        // History ring buffer update
        "DB_Production".Hist_Index := "DB_Production".Hist_Index + 1;
        IF "DB_Production".Hist_Index > 100 THEN
            "DB_Production".Hist_Index := 1;
        END_IF;
        IF "DB_Production".Hist_Count < 100 THEN
            "DB_Production".Hist_Count := "DB_Production".Hist_Count + 1;
        END_IF;
        "DB_Production".Hist_Result["DB_Production".Hist_Index] := "DB_Production".LastResult;
        "DB_Production".Hist_Program["DB_Production".Hist_Index] := "DB_Production".LastProgram;
        "DB_Production".Hist_Duration_s["DB_Production".Hist_Index] := "DB_Production".LastDuration_s;
        "DB_Production".Hist_ErrorCode["DB_Production".Hist_Index] := "DB_Production".LastErrorCode;
        "DB_Production".Hist_ErrorLine["DB_Production".Hist_Index] := "DB_Production".LastErrorLine;
        "DB_Production".Hist_Time["DB_Production".Hist_Index] := #prodTimeNow;
    END_IF;

    // Edge: NOK (enter STATE_ERROR with active cycle)
    IF (#State = STATE_ERROR) AND (#prevState <> STATE_ERROR) AND "DB_Production".CurrentActive THEN
        "DB_Production".LastResult := 2;  // NOK
        "DB_Production".LastProgram := #activeProgram;
        "DB_Production".LastDuration_s := "DB_HMI".ElapsedSeconds;
        "DB_Production".LastErrorCode := #fbAlarmManager.ActiveErrorCode;
        "DB_Production".LastErrorLine := "DB_Diagnostic".Error_Line;
        "DB_Production".TotalNOK := "DB_Production".TotalNOK + 1;
        #prodTimeStatus := RD_SYS_T(OUT => #prodTimeNow);
        "DB_Production".LastEndTime := #prodTimeNow;
        "DB_Production".CurrentActive := FALSE;

        // History ring buffer update
        "DB_Production".Hist_Index := "DB_Production".Hist_Index + 1;
        IF "DB_Production".Hist_Index > 100 THEN
            "DB_Production".Hist_Index := 1;
        END_IF;
        IF "DB_Production".Hist_Count < 100 THEN
            "DB_Production".Hist_Count := "DB_Production".Hist_Count + 1;
        END_IF;
        "DB_Production".Hist_Result["DB_Production".Hist_Index] := "DB_Production".LastResult;
        "DB_Production".Hist_Program["DB_Production".Hist_Index] := "DB_Production".LastProgram;
        "DB_Production".Hist_Duration_s["DB_Production".Hist_Index] := "DB_Production".LastDuration_s;
        "DB_Production".Hist_ErrorCode["DB_Production".Hist_Index] := "DB_Production".LastErrorCode;
        "DB_Production".Hist_ErrorLine["DB_Production".Hist_Index] := "DB_Production".LastErrorLine;
        "DB_Production".Hist_Time["DB_Production".Hist_Index] := #prodTimeNow;
    END_IF;

    // Edge: STOPPED via STOP sequence (STOPPING / STOP_GOHOME / STOP_GOTOZERO → STOPPED)
    IF (#State = STATE_STOPPED) AND
       ((#prevState = STATE_STOPPING) OR (#prevState = STATE_STOP_GOHOME) OR (#prevState = STATE_STOP_GOTOZERO)) AND
       "DB_Production".CurrentActive THEN
        "DB_Production".LastResult := 3;  // STOP
        "DB_Production".LastProgram := #activeProgram;
        "DB_Production".LastDuration_s := "DB_HMI".ElapsedSeconds;
        "DB_Production".LastErrorCode := 0;
        "DB_Production".LastErrorLine := -1;
        "DB_Production".TotalStopped := "DB_Production".TotalStopped + 1;
        #prodTimeStatus := RD_SYS_T(OUT => #prodTimeNow);
        "DB_Production".LastEndTime := #prodTimeNow;
        "DB_Production".CurrentActive := FALSE;

        // History ring buffer update
        "DB_Production".Hist_Index := "DB_Production".Hist_Index + 1;
        IF "DB_Production".Hist_Index > 100 THEN
            "DB_Production".Hist_Index := 1;
        END_IF;
        IF "DB_Production".Hist_Count < 100 THEN
            "DB_Production".Hist_Count := "DB_Production".Hist_Count + 1;
        END_IF;
        "DB_Production".Hist_Result["DB_Production".Hist_Index] := "DB_Production".LastResult;
        "DB_Production".Hist_Program["DB_Production".Hist_Index] := "DB_Production".LastProgram;
        "DB_Production".Hist_Duration_s["DB_Production".Hist_Index] := "DB_Production".LastDuration_s;
        "DB_Production".Hist_ErrorCode["DB_Production".Hist_Index] := "DB_Production".LastErrorCode;
        "DB_Production".Hist_ErrorLine["DB_Production".Hist_Index] := "DB_Production".LastErrorLine;
        "DB_Production".Hist_Time["DB_Production".Hist_Index] := #prodTimeNow;
    END_IF;

    // Production RESET: clear counters + history
    IF #prodResetEdge THEN
        "DB_Production".TotalStarted := 0;
        "DB_Production".TotalOK := 0;
        "DB_Production".TotalNOK := 0;
        "DB_Production".TotalStopped := 0;
        "DB_Production".Hist_Index := 0;
        "DB_Production".Hist_Count := 0;
        // Optionally also clear last cycle summary
        "DB_Production".LastResult := 0;
        "DB_Production".LastProgram := 0;
        "DB_Production".LastDuration_s := 0;
        "DB_Production".LastErrorCode := 0;
        "DB_Production".LastErrorLine := -1;
        "DB_Production".CurrentActive := FALSE;
    END_IF;

    // Last-cycle RESET: only clear last cycle summary (counters and history are preserved)
    IF #lastCycleResetEdge THEN
        "DB_Production".LastResult := 0;
        "DB_Production".LastProgram := 0;
        "DB_Production".LastDuration_s := 0;
        "DB_Production".LastErrorCode := 0;
        "DB_Production".LastErrorLine := -1;
    END_IF;

    // Update prevState for next cycle
    #prevState := #State;

    // =========================================================================
    // RECIPE HANDLER - Execute based on active program
    // =========================================================================
    CASE #activeProgram OF
        1: #fbRecipeHandler(Start := #bStartSeq, Stop := #fbInputs.Cmd_Stop,
                            Pause := #bPauseActive, Reset := #fbInputs.Cmd_Reset OR #bResetRecipe,
                            StartLine := MAX(IN1:= INT#0, IN2:= #savedLineIndex),
                            LineCount := #activeLineCount,
                            Lines := "DB_RecipeProgram1".Lines,
                            Axis_X := #Axis_X, Axis_Z := #Axis_Z);
        2: #fbRecipeHandler(Start := #bStartSeq, Stop := #fbInputs.Cmd_Stop,
                            Pause := #bPauseActive, Reset := #fbInputs.Cmd_Reset OR #bResetRecipe,
                            StartLine := MAX(IN1:= INT#0,IN2:= #savedLineIndex),
                            LineCount := #activeLineCount,
                            Lines := "DB_RecipeProgram2".Lines,
                            Axis_X := #Axis_X, Axis_Z := #Axis_Z);
        3: #fbRecipeHandler(Start := #bStartSeq, Stop := #fbInputs.Cmd_Stop,
                            Pause := #bPauseActive, Reset := #fbInputs.Cmd_Reset OR #bResetRecipe,
                            StartLine := MAX(IN1:= INT#0,IN2:= #savedLineIndex),
                            LineCount := #activeLineCount,
                            Lines := "DB_RecipeProgram3".Lines,
                            Axis_X := #Axis_X, Axis_Z := #Axis_Z);
        4: #fbRecipeHandler(Start := #bStartSeq, Stop := #fbInputs.Cmd_Stop,
                            Pause := #bPauseActive, Reset := #fbInputs.Cmd_Reset OR #bResetRecipe,
                            StartLine := MAX(IN1:= INT#0,IN2:= #savedLineIndex),
                            LineCount := #activeLineCount,
                            Lines := "DB_RecipeProgram4".Lines,
                            Axis_X := #Axis_X, Axis_Z := #Axis_Z);
        5: #fbRecipeHandler(Start := #bStartSeq, Stop := #fbInputs.Cmd_Stop,
                            Pause := #bPauseActive, Reset := #fbInputs.Cmd_Reset OR #bResetRecipe,
                            StartLine := MAX(IN1:= INT#0,IN2:= #savedLineIndex),
                            LineCount := #activeLineCount,
                            Lines := "DB_RecipeProgram5".Lines,
                            Axis_X := #Axis_X, Axis_Z := #Axis_Z);
    END_CASE;

    // Homing -- sequential pattern: STATE_HOMING (startup) and STATE_STOP_GOHOME (post-stop)
    // both use homeSeqState + bHomeXExec/bHomeZExec.
    // Mode SEL: mode 3 (active+zero) is forced in STATE_HOMING; other states use DB_Manual.HomingMode.
    #fbHomeX(
        Execute := #bHomeXExec,
        Mode := SEL(G := (#State = STATE_HOMING AND #bHomeXExec), IN0 := 3, IN1 := "DB_Manual".HomingMode),
        Position := "DB_MachineConfig".HomeOffset_X,
        Axis := #Axis_X
    );
    #fbHomeZ(
        Execute := #bHomeZExec,
        Mode := SEL(G := (#State = STATE_HOMING AND #bHomeZExec), IN0 := 3, IN1 := "DB_Manual".HomingMode),
        Position := "DB_MachineConfig".HomeOffset_Z,
        Axis := #Axis_Z
    );
    #fbHomeTool(
        Execute  := #bHomeToolExec,
        Mode     := SEL(G := (#State = STATE_HOMING AND #bHomeToolExec), IN0 := 3, IN1 := "DB_Manual".HomingMode),
        Position := 0.0,
        Axis     := #Axis_Tool
    );
    // PNP halt FBs: Execute stays TRUE until bHaltX/Z_PNP is cleared (on return to STATE_STOPPED)
    #fbHaltX_PNP(Execute := #bHaltX_PNP, Axis := #Axis_X);
    #fbHaltZ_PNP(Execute := #bHaltZ_PNP, Axis := #Axis_Z);

    // Tool changer -- only rotates the turret; axis positioning done by G-code
    #fbToolChanger(Execute := #bToolExecute, ToolNumber := #activeToolReq,
                   Axis_Tool := #Axis_Tool);

    // Motion FBs for moving to position 0 after stop
    #fbMoveX_Stop(Execute := #bStopMoveX, Position := 0.0, Velocity := "DB_MachineConfig".RapidVelocity, Axis := #Axis_X);
    #fbMoveZ_Stop(Execute := #bStopMoveZ, Position := 0.0, Velocity := "DB_MachineConfig".RapidVelocity, Axis := #Axis_Z);
    // Homing clearance moves -- pre (clear PNP zone) and post (move away after homing)
    // Target: HomeOffset + PostHome_Clearance (outside PNP sensor range)
    #fbMoveX_HomeClr(Execute  := #bHomeClrX,
                     Position := "DB_MachineConfig".HomeOffset_X + "DB_MachineConfig".PostHome_Clearance,
                     Velocity := "DB_MachineConfig".HomeVelocity,
                     Axis     := #Axis_X);
    #fbMoveZ_HomeClr(Execute  := #bHomeClrZ,
                     Position := "DB_MachineConfig".HomeOffset_Z + "DB_MachineConfig".PostHome_Clearance,
                     Velocity := "DB_MachineConfig".HomeVelocity,
                     Axis     := #Axis_Z);

    // Manual mode - sync aliases first
    // In STATE_PNP_HALT: block jog direction that would drive the axis deeper into the PNP zone.
    // Jog toward the active PNP zone is blocked; jog away (escape direction) is passed through.
    IF #State = STATE_PNP_HALT THEN
        "DB_Manual".Jog_Plus  := "DB_Manual".Btn_JogPlus AND NOT (
            ("DB_Manual".SelectedAxis = 0 AND #HW_PNP_X_Max) OR
            ("DB_Manual".SelectedAxis = 1 AND #HW_PNP_Z_Max));
        "DB_Manual".Jog_Minus := "DB_Manual".Btn_JogMinus AND NOT (
            ("DB_Manual".SelectedAxis = 0 AND #HW_PNP_X_Min) OR
            ("DB_Manual".SelectedAxis = 1 AND #HW_PNP_Z_Min));
    ELSE
        "DB_Manual".Jog_Plus  := "DB_Manual".Btn_JogPlus;
        "DB_Manual".Jog_Minus := "DB_Manual".Btn_JogMinus;
    END_IF;
    "DB_Manual".Btn_HomeAxis := "DB_Manual".Btn_Home;

    #fbManualMode(Enable := (#State = STATE_MANUAL OR #State = STATE_PNP_HALT),
                  SelectedAxis := "DB_Manual".SelectedAxis,
                  Jog_Plus := "DB_Manual".Jog_Plus, Jog_Minus := "DB_Manual".Jog_Minus,
                  JogSpeed := "DB_Manual".JogSpeed,
                  MoveAbsolute := "DB_Manual".Btn_MoveAbsolute, TargetPosition := "DB_Manual".MoveToPosition,
                  HomeAxis := "DB_Manual".Btn_HomeAxis, HomeAll := "DB_Manual".Btn_HomeAll,
                  HomingMode := "DB_Manual".HomingMode, HomePosition := 0.0,
                  GoSafe := "DB_Manual".Btn_GoSafe, GoZero := "DB_Manual".Btn_GoZero,
                  SafeToJog := #fbSafetyMonitor.SafeToJog, Reset := #fbInputs.Cmd_Reset,
                  PNP_X_Min := #HW_PNP_X_Min, PNP_Z_Min := #HW_PNP_Z_Min,
                  ToolStepCW := "DB_Manual".Btn_ToolStepCW, ToolStepCCW := "DB_Manual".Btn_ToolStepCCW,
                  ToolStepAngle := "DB_Manual".ToolStepAngle, ToolStepSpeed := "DB_Manual".ToolStepSpeed,
                  Axis_X := #Axis_X, Axis_Z := #Axis_Z, Axis_Tool := #Axis_Tool, Axis_Spindle := #Axis_Spindle);

    // Update manual mode status
    "DB_Manual".JogBusy := #fbManualMode.Busy;
    "DB_Manual".ManualBusy := #fbManualMode.Busy;       // Alias
    "DB_Manual".JogError := #fbManualMode.Error;
    "DB_Manual".ManualError := #fbManualMode.Error;     // Alias
    "DB_Manual".JogErrorID := #fbManualMode.ErrorID;
    "DB_Manual".ManualErrorID := #fbManualMode.ErrorID; // Alias
    "DB_Manual".SelectedAxisPos := SEL(G := "DB_Manual".SelectedAxis = 0,
                                        IN0 := #Axis_Z.ActualPosition, IN1 := #Axis_X.ActualPosition);
    "DB_Manual".SelectedAxisName := SEL(G := "DB_Manual".SelectedAxis = 0, IN0 := 'Z', IN1 := 'X');
    "DB_Manual".ToolPosition := #Axis_Tool.ActualPosition;
    "DB_Manual".ActiveAxis := #fbManualMode.ActiveAxis;

    // Forward manual mode errors to alarm manager (once, on rising edge)
    IF #fbManualMode.Error AND NOT #prevManualError THEN
        #newErrorFlag := TRUE;
        #newErrorCode := #fbManualMode.ErrorID;
        // DB_HMI.ErrorDetail is written directly inside FB_ManualMode at each error point.
        // Write ErrorText here as a fallback for any code not yet handled with direct detail.
        "DB_HMI".ErrorText := 'Manual mode error - check ErrorDetail and ErrorID';
    END_IF;
    #prevManualError := #fbManualMode.Error;

    // =========================================================================
    // SPINDLE CONTROL
    // Manual mode spindle control via DB_Manual buttons
    // Recipe handler spindle control via bSpindleStart/bSpindleStop flags
    // =========================================================================
    #fbSpindleControl(
        Enable := #bDrivesEnable,  // Drive stays powered during normal operation; cut on E-Stop or STATE_ERROR
        Start := "DB_Manual".Btn_SpindleStart OR #bSpindleStart,
        Stop := "DB_Manual".Btn_SpindleStop OR #bSpindleStop OR #fbInputs.Cmd_Stop,
        SetSpeed := SEL(G := (#State = STATE_MANUAL),
                        IN0 := "DB_Spindle".Cmd_SetSpeed,
                        IN1 := "DB_Manual".Manual_SpindleSpeed),
        Direction := SEL(G := (#State = STATE_MANUAL),
                         IN0 := "DB_Spindle".Cmd_Direction,
                         IN1 := "DB_Manual".Manual_SpindleDir),
        SpeedOverride := "DB_Spindle".SpeedOverride,
        Reset := #fbInputs.Cmd_Reset OR #bResetRecipe,  // Also reset on recipe restart (clears state 999 error)
        AckError := #ackEdge OR "DB_Manual".Btn_SpindleAckError,  // Main Ack or spindle-specific Ack (no full Reset needed)
        Axis_Spindle := #Axis_Spindle
    );

    // Diagnostic output
    "DB_Diagnostic".Process_State        := #State;
    "DB_Diagnostic".Process_SafeToRun    := #SafeToRun;
    "DB_Diagnostic".Process_DrivesEnable := #bDrivesEnable;
    "DB_Diagnostic".Recipe_CurrentProgram := #activeProgram;
    "DB_Diagnostic".Recipe_TotalLines    := #activeLineCount;
    "DB_Diagnostic".Axis_X_Pos           := #Axis_X.ActualPosition;
    "DB_Diagnostic".Axis_Z_Pos           := #Axis_Z.ActualPosition;
    "DB_Diagnostic".Axis_X_Enabled       := #fbPowerX.Status;
    "DB_Diagnostic".Axis_Z_Enabled       := #fbPowerZ.Status;
    "DB_Diagnostic".Axis_X_Homed         := #Axis_X.StatusBits.HomingDone;
    "DB_Diagnostic".Axis_Z_Homed         := #Axis_Z.StatusBits.HomingDone;

    // =========================================================================
    // CONTACTOR CONTROL -- called as the last step of FB_Process.
    // FC_ContactorControl reads DB_HMI.Btn_Contactor_* and Bypass_EStop/HasError.
    // In auto mode STATE_STARTING already sets these flags TRUE; they are reflected to I/O here.
    // Called here rather than from OB1 to ensure contactor logic runs in sync with the process.
    // =========================================================================
    "FC_ContactorControl"();
END_FUNCTION_BLOCK
